// TIA Portal V19 export
TYPE "LEXCHANGETRAY_typeHandlingXyzEm_toNgConveyoReq"
// stored: Access Published
   STRUCT
      transferEnable : Bool;   // 请求转移
      ngCellsCounts : Int;   // NG电池数量
   END_STRUCT;
END_TYPE
